Fanuc KAREL source: IO0193.KL

PROGRAM IO0193
%NOLOCKGROUP
ROUTINE RTEST
VAR
L1 : ARRAY[3] OF INTEGER;L2 : XYZWPR
L3 : JOINTPOS9
L4 : POSITION
A:BOOLEAN
S1:INTEGER
B:REAL
C:BOOLEAN
D:REAL
BEGIN
--
--
A=TRUE
L1[1]=2
C=TRUE
D=1.0
L2=GET_POS_REG(1,S1,1)
END RTEST
BEGIN
RTEST
END IO0193
